FUNCTION_BLOCK DrillController
  (* Standard: 61499-2 *)
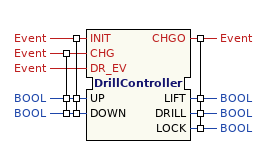
  EVENT_INPUT
    INIT WITH UP, DOWN;
    CHG WITH UP, DOWN;
    DR_EV;
  END_EVENT
  EVENT_OUTPUT
    CHGO WITH LIFT, DRILL, LOCK;
  END_EVENT
  VAR_INPUT
    UP : BOOL;
    DOWN : BOOL;
  END_VAR
  VAR_OUTPUT
    LIFT : BOOL;
    DRILL : BOOL;
    LOCK : BOOL;
  END_VAR
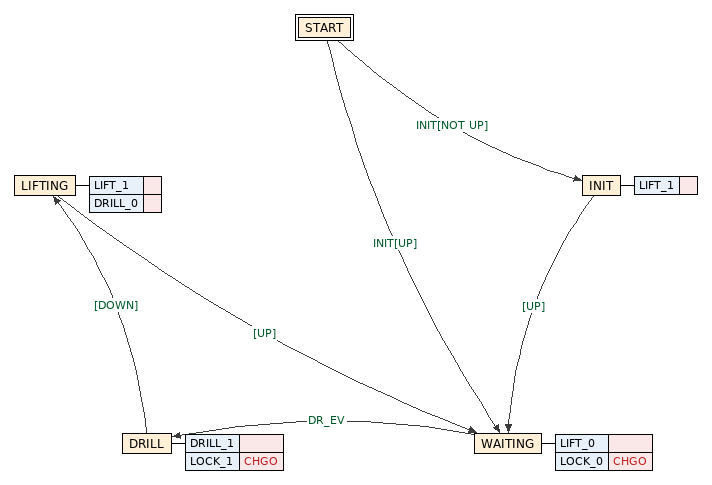
  EC_STATES
    START;
    INIT : LIFT_1;
    WAITING : LIFT_0, LOCK_0 -> CHGO;
    DRILL : DRILL_1, LOCK_1 -> CHGO;
    LIFTING : LIFT_1, DRILL_0;
  END_STATES
  EC_TRANSITIONS
    START TO INIT := INIT[NOT UP];
    INIT TO WAITING := [UP];
    START TO WAITING := INIT[UP];
    WAITING TO DRILL := DR_EV;
    DRILL TO LIFTING := [DOWN];
    LIFTING TO WAITING := [UP];
  END_TRANSITIONS
  ALGORITHM LIFT_0 IN ST:
LIFT := FALSE;&#10;
  END_ALGORITHM
  ALGORITHM LIFT_1 IN ST:
LIFT := TRUE;&#10;
  END_ALGORITHM
  ALGORITHM DRILL_0 IN ST:
DRILL := FALSE;&#10;
  END_ALGORITHM
  ALGORITHM DRILL_1 IN ST:
DRILL := TRUE;&#10;
  END_ALGORITHM
  ALGORITHM LOCK_0 IN ST:
LOCK := FALSE;&#10;
  END_ALGORITHM
  ALGORITHM LOCK_1 IN ST:
LOCK := TRUE;&#10;
  END_ALGORITHM
END_FUNCTION_BLOCK
